Staubli VAL3: interfaceCS8.pjx

--- interfaceCS8.pjx ---
Parameters version=s7.11 stackSize=5000 millimeterUnit=true
Program file=ack.pgx
Program file=clearScreen.pgx
Program file=debug.pgx
Program file=feedbackStatus.pgx
Program file=init.pgx
Program file=motionBuffer.pgx
Program file=motionProgress.pgx
Program file=motionStatus.pgx
Program file=start.pgx
Program file=stop.pgx
Program file=trajBuffer.pgx
Program file=velOverwrite.pgx
Data file=interfaceCS8.dtx
Library alias=libQueueFuncs path=Disk://ros_libs/QueueFuncs/QueueFuncs.pjx

--- cartStatus.pgx ---
public program cartStatus(num x_nCartConnFlag, num x_nLastMsgAge)
begin

  // update connection status on port 11001 (cartesian server)

  gotoxy(scMonitor, 0,1)
  put(scMonitor, "Port 11001:")
  gotoxy(scMonitor, 12,1)
  switch x_nCartConnFlag
    case -1
      put(scMonitor, "connection lost")
    break
    case 0
      put(scMonitor, "not connected")
    break
    case 1
      put(scMonitor, "connected")
    break
    default
      put(scMonitor, "not connected")
    break
  endSwitch

  gotoxy(scMonitor, 0,2)
  put(scMonitor, "Last cart msg:")
  gotoxy(scMonitor, 14,2)
  if (x_nLastMsgAge < 0)
    put(scMonitor, "n/a")
  else
    put(scMonitor, toString(".1", x_nLastMsgAge) + " s")
  endIf

end

--- feedbackStatus.pgx ---
public program feedbackStatus(num x_nOutConnFlag)
begin

  // update connection status on port 11002 (feedback server)

  gotoxy(scMonitor, 0,3)
  // 11 characters: gotoxy(12,3) to insert status
  put(scMonitor, "Port 11002:")
  gotoxy(scMonitor, 12,3)
  switch x_nOutConnFlag
    case -1
      put(scMonitor, "connection lost")
    break
    case 0
      put(scMonitor, "not connected")
    break
    case 1
      put(scMonitor, "connected")
    break
    default
      put(scMonitor, "not connected")
    break
  endSwitch

end
